Fanuc KAREL source: kd00003.KL

-- PROVISIONAL review KL for V940-1; original PC SHA256 6b737f8f8bea17363a8d6c4f77ae3a2ff3bcef3cfa63abb60832ba8835f21295
-- Incomplete behavior may be omitted. Consult companion uncertainty JSON. Do not deploy.
PROGRAM KD00003
%NOLOCKGROUP
-- UNRESOLVED_DECL I type=fd0010
-- UNRESOLVED_DECL J type=fd0010
-- UNRESOLVED_DECL B type=fd0012
-- UNRESOLVED_DECL R type=fd0011
-- UNRESOLVED_DECL S type=fd1f50
BEGIN
  -- V9_ZERO_TABLE_METADATA_HINT layout=0001; no indexed target words; source/name/runtime held
  -- UNRESOLVED_PC offsets 5-12; opcodes 9D,23
  -- UNRESOLVED_PC offsets 17-21; opcodes 7F
END KD00003
